// TIA Portal V17 export
// export: Created 2024-09-27T18:53:46.9042385Z, ExportSetting WithDefaults, DisplayName Totally Integrated Automation Portal, DisplayVersion V17, DisplayName TIA Portal Openness, DisplayVersion V17, DisplayName TIA Portal Version Control Interface, DisplayVersion V17, DisplayName STEP 7 Professional, DisplayVersion V17, DisplayName STEP 7 Safety, DisplayVersion V17, DisplayName WinCC Professional, DisplayVersion V17
FUNCTION "AUTOMAT" : Void   // FC6, LAD
{ S7_Optimized_Access := 'TRUE' }
VERSION : 0.1
// stored: AutoNumber true, IsIECCheckEnabled false, SetENOAutomatically false, UDAEnableTagReadback false
   VAR_TEMP
      m_zbocze_czujnik_poz_odb_stoł : Bool;
      m_zbocze_czujnik_stołP : Bool;
      m_zboczeN_czuj_plyt_przód : Bool;
      m_memo_stol_poz : Bool;
   END_VAR
   VAR_TEMP   // added for the SCL form of the ladder/FBD networks
      _w1 : Bool;
      _w2 : Bool;
   END_VAR
BEGIN

REGION Network 1: CHECK SERVO CONDITIONS
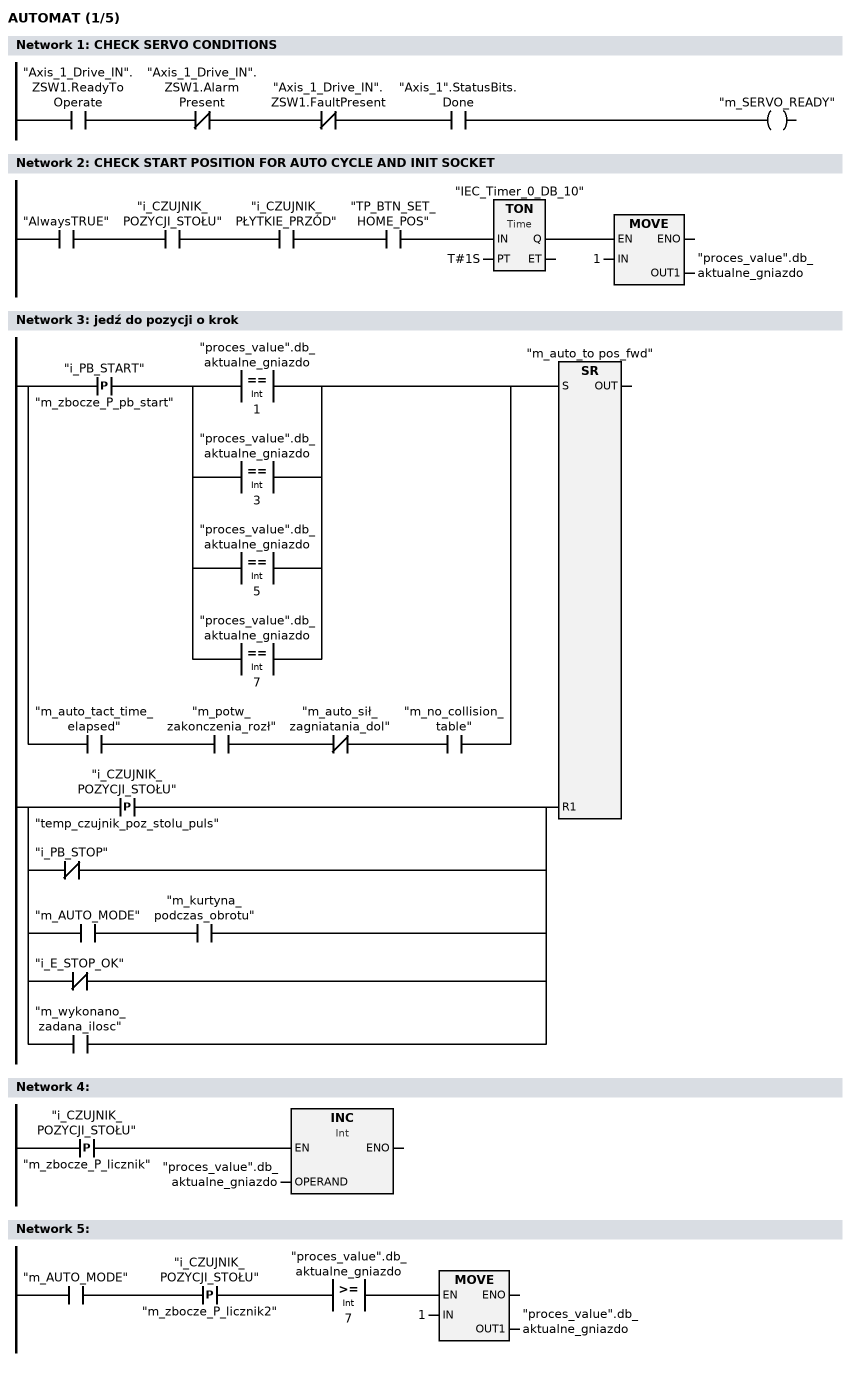
   RUNG wire#powerrail
      Contact( "Axis_1_Drive_IN".ZSW1.ReadyToOperate )
      I_Contact( "Axis_1_Drive_IN".ZSW1.AlarmPresent )
      I_Contact( "Axis_1_Drive_IN".ZSW1.FaultPresent )
      Contact( "Axis_1".StatusBits.Done )
      Coil( "m_SERVO_READY" )
   END_RUNG
   // the same network as SCL:
   "m_SERVO_READY" := "Axis_1_Drive_IN".ZSW1.ReadyToOperate AND NOT "Axis_1_Drive_IN".ZSW1.AlarmPresent AND NOT "Axis_1_Drive_IN".ZSW1.FaultPresent AND "Axis_1".StatusBits.Done;
END_REGION

REGION Network 2: CHECK START POSITION FOR AUTO CYCLE AND INIT SOCKET
   RUNG wire#powerrail
      Contact( "AlwaysTRUE" )
      Contact( "i_CZUJNIK_POZYCJI_STOŁU" )
      Contact( "i_CZUJNIK_PŁYTKIE_PRZÓD" )
      Contact( "TP_BTN_SET_HOME_POS" )
      { S7_Templates := "time_type := Time" } "IEC_Timer_0_DB_10".TON(pt := T#1S, et =>)
      Move(in := 1, out1 => "proces_value".db_aktualne_gniazdo)
   END_RUNG
   // the same network as SCL:
   "IEC_Timer_0_DB_10".TON(IN := "AlwaysTRUE" AND "i_CZUJNIK_POZYCJI_STOŁU" AND "i_CZUJNIK_PŁYTKIE_PRZÓD" AND "TP_BTN_SET_HOME_POS",
                           PT := T#1S);
   IF "IEC_Timer_0_DB_10".Q THEN "proces_value".db_aktualne_gniazdo := 1; END_IF;
END_REGION

REGION Network 3: jedź do pozycji o krok
   RUNG wire#powerrail
      P_Contact(operand := "i_PB_START", bit := "m_zbocze_P_pb_start")
      wire#w1
      { S7_Templates := "SrcType := Int" } EQ_Contact(in1 := "proces_value".db_aktualne_gniazdo, in2 := 1)
      wire#w2
      S_SR(operand := "m_auto_to pos_fwd", r1 := wire#w3)
   END_RUNG
   RUNG wire#w1
      { S7_Templates := "SrcType := Int" } EQ_Contact(in1 := "proces_value".db_aktualne_gniazdo, in2 := 3)
   END_RUNG wire#w2
   RUNG wire#w1
      { S7_Templates := "SrcType := Int" } EQ_Contact(in1 := "proces_value".db_aktualne_gniazdo, in2 := 5)
   END_RUNG wire#w2
   RUNG wire#w1
      { S7_Templates := "SrcType := Int" } EQ_Contact(in1 := "proces_value".db_aktualne_gniazdo, in2 := 7)
   END_RUNG wire#w2
   RUNG wire#powerrail
      Contact( "m_auto_tact_time_elapsed" )
      Contact( "m_potw_zakonczenia_rozł" )
      I_Contact( "m_auto_sił_zagniatania_dol" )
      Contact( "m_no_collision_table" )
   END_RUNG wire#w2
   RUNG wire#powerrail
      P_Contact(operand := "i_CZUJNIK_POZYCJI_STOŁU", bit := "temp_czujnik_poz_stolu_puls")
   END_RUNG wire#w3
   RUNG wire#powerrail
      I_Contact( "i_PB_STOP" )
   END_RUNG wire#w3
   RUNG wire#powerrail
      Contact( "m_AUTO_MODE" )
      Contact( "m_kurtyna_podczas_obrotu" )
   END_RUNG wire#w3
   RUNG wire#powerrail
      I_Contact( "i_E_STOP_OK" )
   END_RUNG wire#w3
   RUNG wire#powerrail
      Contact( "m_wykonano_zadana_ilosc" )
   END_RUNG wire#w3
   // the same network as SCL:
   #_w1 := "i_PB_START" AND NOT "m_zbocze_P_pb_start";   // rising edge of "i_PB_START"
   "m_zbocze_P_pb_start" := "i_PB_START";
   #_w2 := "i_CZUJNIK_POZYCJI_STOŁU" AND NOT "temp_czujnik_poz_stolu_puls";   // rising edge of "i_CZUJNIK_POZYCJI_STOŁU"
   "temp_czujnik_poz_stolu_puls" := "i_CZUJNIK_POZYCJI_STOŁU";
   IF (#_w1 AND (("proces_value".db_aktualne_gniazdo = 1) OR ("proces_value".db_aktualne_gniazdo = 3) OR ("proces_value".db_aktualne_gniazdo = 5) OR ("proces_value".db_aktualne_gniazdo = 7))) OR ("m_auto_tact_time_elapsed" AND "m_potw_zakonczenia_rozł" AND NOT "m_auto_sił_zagniatania_dol" AND "m_no_collision_table") THEN
       "m_auto_to pos_fwd" := TRUE;   // SR flip-flop
   END_IF;
   IF #_w2 OR NOT "i_PB_STOP" OR ("m_AUTO_MODE" AND "m_kurtyna_podczas_obrotu") OR NOT "i_E_STOP_OK" OR "m_wykonano_zadana_ilosc" THEN
       "m_auto_to pos_fwd" := FALSE;
   END_IF;
END_REGION

REGION Network 4
   RUNG wire#powerrail
      P_Contact(operand := "i_CZUJNIK_POZYCJI_STOŁU", bit := "m_zbocze_P_licznik")
      { S7_Templates := "DestType := Int" } Inc( "proces_value".db_aktualne_gniazdo )
   END_RUNG
   // the same network as SCL:
   #_w1 := "i_CZUJNIK_POZYCJI_STOŁU" AND NOT "m_zbocze_P_licznik";   // rising edge of "i_CZUJNIK_POZYCJI_STOŁU"
   "m_zbocze_P_licznik" := "i_CZUJNIK_POZYCJI_STOŁU";
   IF #_w1 THEN "proces_value".db_aktualne_gniazdo := "proces_value".db_aktualne_gniazdo + 1; END_IF;
END_REGION

REGION Network 5
   RUNG wire#powerrail
      Contact( "m_AUTO_MODE" )
      P_Contact(operand := "i_CZUJNIK_POZYCJI_STOŁU", bit := "m_zbocze_P_licznik2")
      { S7_Templates := "SrcType := Int" } GE_Contact(in1 := "proces_value".db_aktualne_gniazdo, in2 := 7)
      Move(in := 1, out1 => "proces_value".db_aktualne_gniazdo)
   END_RUNG
   // the same network as SCL:
   #_w1 := "m_AUTO_MODE" AND "i_CZUJNIK_POZYCJI_STOŁU" AND NOT "m_zbocze_P_licznik2";   // rising edge of "i_CZUJNIK_POZYCJI_STOŁU"
   "m_zbocze_P_licznik2" := "i_CZUJNIK_POZYCJI_STOŁU";
   IF #_w1 AND ("proces_value".db_aktualne_gniazdo >= 7) THEN
       "proces_value".db_aktualne_gniazdo := 1;
   END_IF;
END_REGION

REGION Network 6: zwłoka taktu
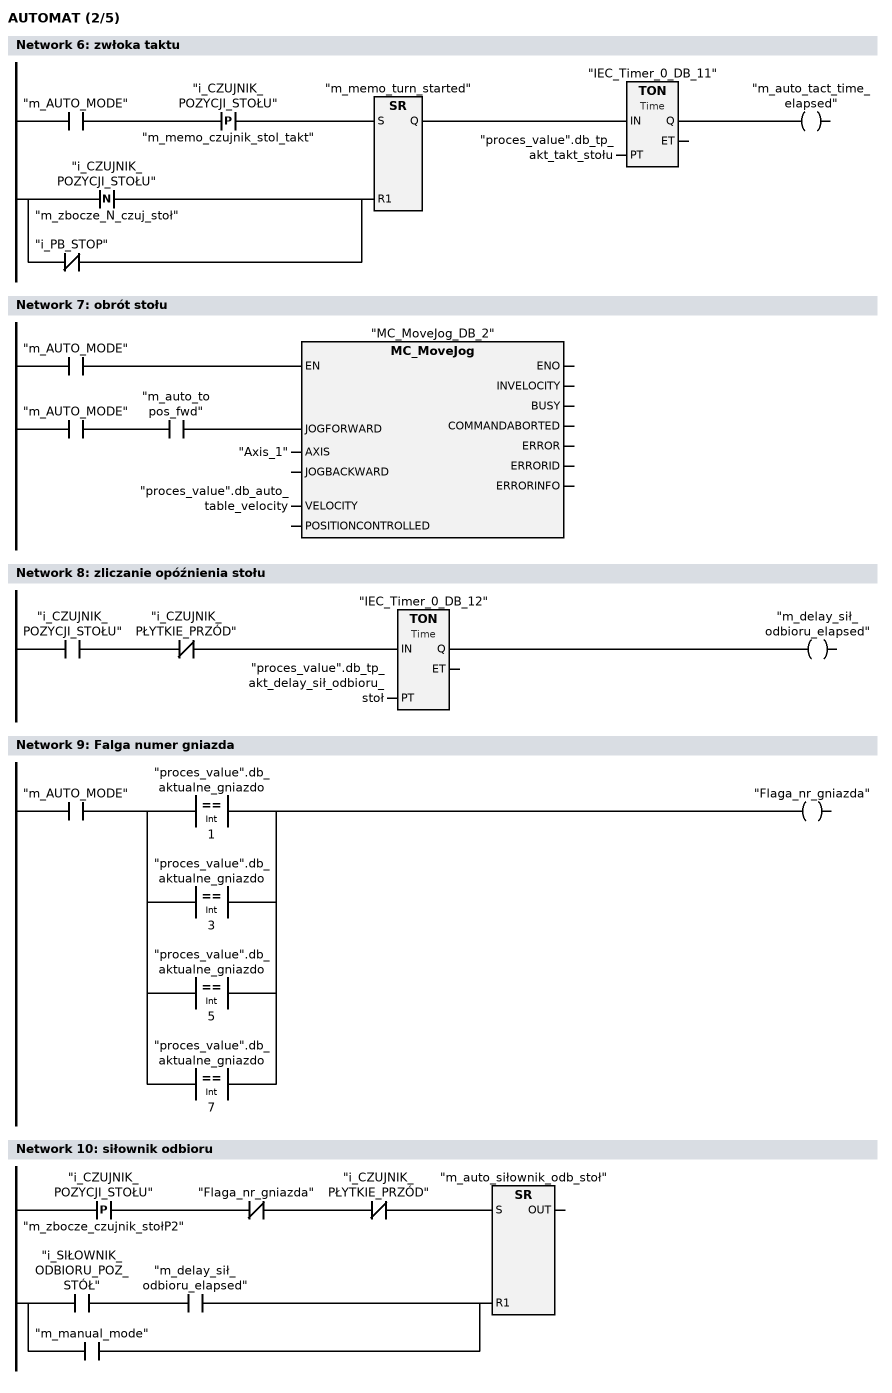
   RUNG wire#powerrail
      Contact( "m_AUTO_MODE" )
      P_Contact(operand := "i_CZUJNIK_POZYCJI_STOŁU", bit := "m_memo_czujnik_stol_takt")
      S_SR(operand := "m_memo_turn_started", r1 := wire#w1)
      { S7_Templates := "time_type := Time" } "IEC_Timer_0_DB_11".TON(pt := "proces_value".db_tp_akt_takt_stołu, et =>)
      Coil( "m_auto_tact_time_elapsed" )
   END_RUNG
   RUNG wire#powerrail
      N_Contact(operand := "i_CZUJNIK_POZYCJI_STOŁU", bit := "m_zbocze_N_czuj_stoł")
   END_RUNG wire#w1
   RUNG wire#powerrail
      I_Contact( "i_PB_STOP" )
   END_RUNG wire#w1
   // the same network as SCL:
   #_w1 := "m_AUTO_MODE" AND "i_CZUJNIK_POZYCJI_STOŁU" AND NOT "m_memo_czujnik_stol_takt";   // rising edge of "i_CZUJNIK_POZYCJI_STOŁU"
   "m_memo_czujnik_stol_takt" := "i_CZUJNIK_POZYCJI_STOŁU";
   #_w2 := NOT "i_CZUJNIK_POZYCJI_STOŁU" AND "m_zbocze_N_czuj_stoł";   // falling edge of "i_CZUJNIK_POZYCJI_STOŁU"
   "m_zbocze_N_czuj_stoł" := "i_CZUJNIK_POZYCJI_STOŁU";
   IF #_w1 THEN
       "m_memo_turn_started" := TRUE;   // SR flip-flop
   END_IF;
   IF #_w2 OR NOT "i_PB_STOP" THEN "m_memo_turn_started" := FALSE; END_IF;
   "IEC_Timer_0_DB_11".TON(IN := "m_memo_turn_started", PT := "proces_value".db_tp_akt_takt_stołu);
   "m_auto_tact_time_elapsed" := "IEC_Timer_0_DB_11".Q;
END_REGION

REGION Network 7: obrót stołu
   RUNG wire#powerrail
      Contact( "m_AUTO_MODE" )
      "MC_MoveJog_DB_2".MC_MoveJog(JogForward := wire#w1, Axis := "Axis_1", JogBackward :=, Velocity := "proces_value".db_auto_table_velocity, PositionControlled :=, InVelocity =>, Busy =>, CommandAborted =>, Error =>, ErrorID =>, ErrorInfo =>)
   END_RUNG
   RUNG wire#powerrail
      Contact( "m_AUTO_MODE" )
      Contact( "m_auto_to pos_fwd" )
   END_RUNG wire#w1
   // the same network as SCL:
   IF "m_AUTO_MODE" THEN
       "MC_MoveJog_DB_2"(JogForward := "m_AUTO_MODE" AND "m_auto_to pos_fwd",   // MC_MoveJog
                         Axis := "Axis_1",
                         Velocity := "proces_value".db_auto_table_velocity);
   END_IF;
END_REGION

REGION Network 8: zliczanie opóźnienia stołu
   RUNG wire#powerrail
      Contact( "i_CZUJNIK_POZYCJI_STOŁU" )
      I_Contact( "i_CZUJNIK_PŁYTKIE_PRZÓD" )
      { S7_Templates := "time_type := Time" } "IEC_Timer_0_DB_12".TON(pt := "proces_value".db_tp_akt_delay_sił_odbioru_stoł, et =>)
      Coil( "m_delay_sił_odbioru_elapsed" )
   END_RUNG
   // the same network as SCL:
   "IEC_Timer_0_DB_12".TON(IN := "i_CZUJNIK_POZYCJI_STOŁU" AND NOT "i_CZUJNIK_PŁYTKIE_PRZÓD",
                           PT := "proces_value".db_tp_akt_delay_sił_odbioru_stoł);
   "m_delay_sił_odbioru_elapsed" := "IEC_Timer_0_DB_12".Q;
END_REGION

REGION Network 9: Falga numer gniazda
   RUNG wire#powerrail
      Contact( "m_AUTO_MODE" )
      wire#w1
      { S7_Templates := "SrcType := Int" } EQ_Contact(in1 := "proces_value".db_aktualne_gniazdo, in2 := 1)
      wire#w2
      Coil( "Flaga_nr_gniazda" )
   END_RUNG
   RUNG wire#w1
      { S7_Templates := "SrcType := Int" } EQ_Contact(in1 := "proces_value".db_aktualne_gniazdo, in2 := 3)
   END_RUNG wire#w2
   RUNG wire#w1
      { S7_Templates := "SrcType := Int" } EQ_Contact(in1 := "proces_value".db_aktualne_gniazdo, in2 := 5)
   END_RUNG wire#w2
   RUNG wire#w1
      { S7_Templates := "SrcType := Int" } EQ_Contact(in1 := "proces_value".db_aktualne_gniazdo, in2 := 7)
   END_RUNG wire#w2
   // the same network as SCL:
   "Flaga_nr_gniazda" := "m_AUTO_MODE" AND (("proces_value".db_aktualne_gniazdo = 1) OR ("proces_value".db_aktualne_gniazdo = 3) OR ("proces_value".db_aktualne_gniazdo = 5) OR ("proces_value".db_aktualne_gniazdo = 7));
END_REGION

REGION Network 10: siłownik odbioru
   RUNG wire#powerrail
      P_Contact(operand := "i_CZUJNIK_POZYCJI_STOŁU", bit := "m_zbocze_czujnik_stołP2")
      I_Contact( "Flaga_nr_gniazda" )
      I_Contact( "i_CZUJNIK_PŁYTKIE_PRZÓD" )
      S_SR(operand := "m_auto_siłownik_odb_stoł", r1 := wire#w1)
   END_RUNG
   RUNG wire#powerrail
      Contact( "i_SIŁOWNIK_ODBIORU_POZ_STÓŁ" )
      Contact( "m_delay_sił_odbioru_elapsed" )
   END_RUNG wire#w1
   RUNG wire#powerrail
      Contact( "m_manual_mode" )
   END_RUNG wire#w1
   // the same network as SCL:
   #_w1 := "i_CZUJNIK_POZYCJI_STOŁU" AND NOT "m_zbocze_czujnik_stołP2";   // rising edge of "i_CZUJNIK_POZYCJI_STOŁU"
   "m_zbocze_czujnik_stołP2" := "i_CZUJNIK_POZYCJI_STOŁU";
   IF #_w1 AND NOT "Flaga_nr_gniazda" AND NOT "i_CZUJNIK_PŁYTKIE_PRZÓD" THEN
       "m_auto_siłownik_odb_stoł" := TRUE;   // SR flip-flop
   END_IF;
   IF ("i_SIŁOWNIK_ODBIORU_POZ_STÓŁ" AND "m_delay_sił_odbioru_elapsed") OR "m_manual_mode" THEN
       "m_auto_siłownik_odb_stoł" := FALSE;
   END_IF;
END_REGION

REGION Network 11
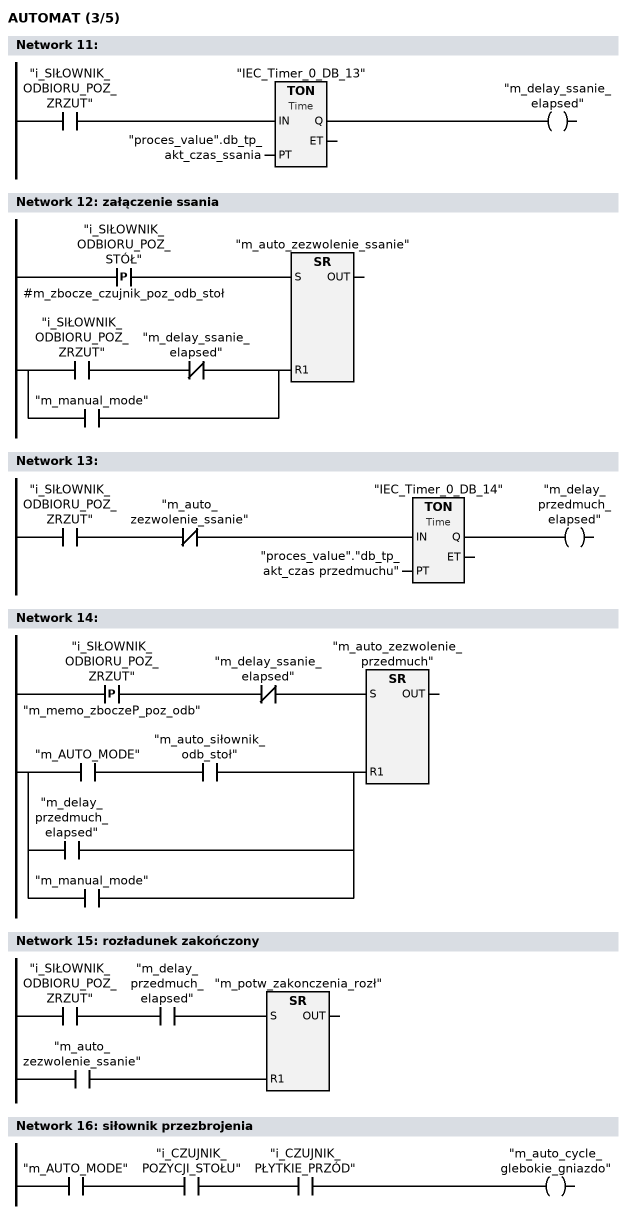
   RUNG wire#powerrail
      Contact( "i_SIŁOWNIK_ODBIORU_POZ_ZRZUT" )
      { S7_Templates := "time_type := Time" } "IEC_Timer_0_DB_13".TON(pt := "proces_value".db_tp_akt_czas_ssania, et =>)
      Coil( "m_delay_ssanie_elapsed" )
   END_RUNG
   // the same network as SCL:
   "IEC_Timer_0_DB_13".TON(IN := "i_SIŁOWNIK_ODBIORU_POZ_ZRZUT", PT := "proces_value".db_tp_akt_czas_ssania);
   "m_delay_ssanie_elapsed" := "IEC_Timer_0_DB_13".Q;
END_REGION

REGION Network 12: załączenie ssania
   RUNG wire#powerrail
      P_Contact(operand := "i_SIŁOWNIK_ODBIORU_POZ_STÓŁ", bit := #m_zbocze_czujnik_poz_odb_stoł)
      S_SR(operand := "m_auto_zezwolenie_ssanie", r1 := wire#w1)
   END_RUNG
   RUNG wire#powerrail
      Contact( "i_SIŁOWNIK_ODBIORU_POZ_ZRZUT" )
      I_Contact( "m_delay_ssanie_elapsed" )
   END_RUNG wire#w1
   RUNG wire#powerrail
      Contact( "m_manual_mode" )
   END_RUNG wire#w1
   // the same network as SCL:
   #_w1 := "i_SIŁOWNIK_ODBIORU_POZ_STÓŁ" AND NOT #m_zbocze_czujnik_poz_odb_stoł;   // rising edge of "i_SIŁOWNIK_ODBIORU_POZ_STÓŁ"
   #m_zbocze_czujnik_poz_odb_stoł := "i_SIŁOWNIK_ODBIORU_POZ_STÓŁ";
   IF #_w1 THEN
       "m_auto_zezwolenie_ssanie" := TRUE;   // SR flip-flop
   END_IF;
   IF ("i_SIŁOWNIK_ODBIORU_POZ_ZRZUT" AND NOT "m_delay_ssanie_elapsed") OR "m_manual_mode" THEN
       "m_auto_zezwolenie_ssanie" := FALSE;
   END_IF;
END_REGION

REGION Network 13
   RUNG wire#powerrail
      Contact( "i_SIŁOWNIK_ODBIORU_POZ_ZRZUT" )
      I_Contact( "m_auto_zezwolenie_ssanie" )
      { S7_Templates := "time_type := Time" } "IEC_Timer_0_DB_14".TON(pt := "proces_value"."db_tp_akt_czas przedmuchu", et =>)
      Coil( "m_delay_przedmuch_elapsed" )
   END_RUNG
   // the same network as SCL:
   "IEC_Timer_0_DB_14".TON(IN := "i_SIŁOWNIK_ODBIORU_POZ_ZRZUT" AND NOT "m_auto_zezwolenie_ssanie",
                           PT := "proces_value"."db_tp_akt_czas przedmuchu");
   "m_delay_przedmuch_elapsed" := "IEC_Timer_0_DB_14".Q;
END_REGION

REGION Network 14
   RUNG wire#powerrail
      P_Contact(operand := "i_SIŁOWNIK_ODBIORU_POZ_ZRZUT", bit := "m_memo_zboczeP_poz_odb")
      I_Contact( "m_delay_ssanie_elapsed" )
      S_SR(operand := "m_auto_zezwolenie_przedmuch", r1 := wire#w1)
   END_RUNG
   RUNG wire#powerrail
      Contact( "m_AUTO_MODE" )
      Contact( "m_auto_siłownik_odb_stoł" )
   END_RUNG wire#w1
   RUNG wire#powerrail
      Contact( "m_delay_przedmuch_elapsed" )
   END_RUNG wire#w1
   RUNG wire#powerrail
      Contact( "m_manual_mode" )
   END_RUNG wire#w1
   // the same network as SCL:
   #_w1 := "i_SIŁOWNIK_ODBIORU_POZ_ZRZUT" AND NOT "m_memo_zboczeP_poz_odb";   // rising edge of "i_SIŁOWNIK_ODBIORU_POZ_ZRZUT"
   "m_memo_zboczeP_poz_odb" := "i_SIŁOWNIK_ODBIORU_POZ_ZRZUT";
   IF #_w1 AND NOT "m_delay_ssanie_elapsed" THEN
       "m_auto_zezwolenie_przedmuch" := TRUE;   // SR flip-flop
   END_IF;
   IF ("m_AUTO_MODE" AND "m_auto_siłownik_odb_stoł") OR "m_delay_przedmuch_elapsed" OR "m_manual_mode" THEN
       "m_auto_zezwolenie_przedmuch" := FALSE;
   END_IF;
END_REGION

REGION Network 15: rozładunek zakończony
   RUNG wire#powerrail
      Contact( "i_SIŁOWNIK_ODBIORU_POZ_ZRZUT" )
      Contact( "m_delay_przedmuch_elapsed" )
      S_SR(operand := "m_potw_zakonczenia_rozł", r1 := wire#w1)
   END_RUNG
   RUNG wire#powerrail
      Contact( "m_auto_zezwolenie_ssanie" )
   END_RUNG wire#w1
   // the same network as SCL:
   IF "i_SIŁOWNIK_ODBIORU_POZ_ZRZUT" AND "m_delay_przedmuch_elapsed" THEN
       "m_potw_zakonczenia_rozł" := TRUE;   // SR flip-flop
   END_IF;
   IF "m_auto_zezwolenie_ssanie" THEN "m_potw_zakonczenia_rozł" := FALSE; END_IF;
END_REGION

REGION Network 16: siłownik przezbrojenia
   RUNG wire#powerrail
      Contact( "m_AUTO_MODE" )
      Contact( "i_CZUJNIK_POZYCJI_STOŁU" )
      Contact( "i_CZUJNIK_PŁYTKIE_PRZÓD" )
      Coil( "m_auto_cycle_glebokie_gniazdo" )
   END_RUNG
   // the same network as SCL:
   "m_auto_cycle_glebokie_gniazdo" := "m_AUTO_MODE" AND "i_CZUJNIK_POZYCJI_STOŁU" AND "i_CZUJNIK_PŁYTKIE_PRZÓD";
END_REGION

REGION Network 17: Interlock na zmiane podczas ruchu siłownika góra dół
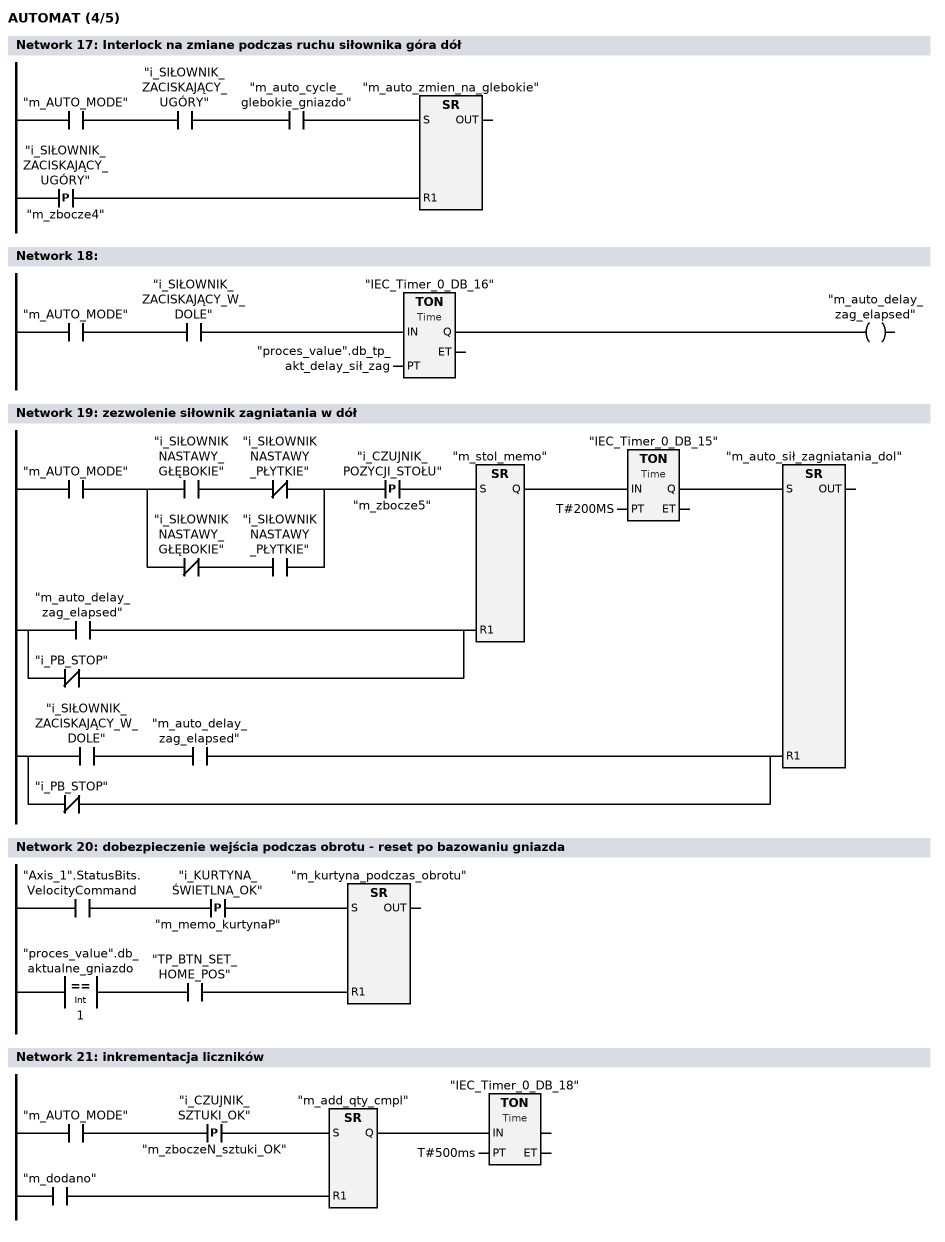
   RUNG wire#powerrail
      Contact( "m_AUTO_MODE" )
      Contact( "i_SIŁOWNIK_ZACISKAJĄCY_UGÓRY" )
      Contact( "m_auto_cycle_glebokie_gniazdo" )
      S_SR(operand := "m_auto_zmien_na_glebokie", r1 := wire#w1)
   END_RUNG
   RUNG wire#powerrail
      P_Contact(operand := "i_SIŁOWNIK_ZACISKAJĄCY_UGÓRY", bit := "m_zbocze4")
   END_RUNG wire#w1
   // the same network as SCL:
   #_w1 := "i_SIŁOWNIK_ZACISKAJĄCY_UGÓRY" AND NOT "m_zbocze4";   // rising edge of "i_SIŁOWNIK_ZACISKAJĄCY_UGÓRY"
   "m_zbocze4" := "i_SIŁOWNIK_ZACISKAJĄCY_UGÓRY";
   IF "m_AUTO_MODE" AND "i_SIŁOWNIK_ZACISKAJĄCY_UGÓRY" AND "m_auto_cycle_glebokie_gniazdo" THEN
       "m_auto_zmien_na_glebokie" := TRUE;   // SR flip-flop
   END_IF;
   IF #_w1 THEN "m_auto_zmien_na_glebokie" := FALSE; END_IF;
END_REGION

REGION Network 18
   RUNG wire#powerrail
      Contact( "m_AUTO_MODE" )
      Contact( "i_SIŁOWNIK_ZACISKAJĄCY_W_DOLE" )
      { S7_Templates := "time_type := Time" } "IEC_Timer_0_DB_16".TON(pt := "proces_value".db_tp_akt_delay_sił_zag, et =>)
      Coil( "m_auto_delay_zag_elapsed" )
   END_RUNG
   // the same network as SCL:
   "IEC_Timer_0_DB_16".TON(IN := "m_AUTO_MODE" AND "i_SIŁOWNIK_ZACISKAJĄCY_W_DOLE",
                           PT := "proces_value".db_tp_akt_delay_sił_zag);
   "m_auto_delay_zag_elapsed" := "IEC_Timer_0_DB_16".Q;
END_REGION

REGION Network 19: zezwolenie siłownik zagniatania w dół
   RUNG wire#powerrail
      Contact( "m_AUTO_MODE" )
      wire#w1
      Contact( "i_SIŁOWNIK NASTAWY_GŁĘBOKIE" )
      I_Contact( "i_SIŁOWNIK NASTAWY _PŁYTKIE" )
      wire#w2
      P_Contact(operand := "i_CZUJNIK_POZYCJI_STOŁU", bit := "m_zbocze5")
      S_SR(operand := "m_stol_memo", r1 := wire#w3)
      { S7_Templates := "time_type := Time" } "IEC_Timer_0_DB_15".TON(pt := T#200MS, et =>)
      S_SR(operand := "m_auto_sił_zagniatania_dol", r1 := wire#w4)
   END_RUNG
   RUNG wire#w1
      I_Contact( "i_SIŁOWNIK NASTAWY_GŁĘBOKIE" )
      Contact( "i_SIŁOWNIK NASTAWY _PŁYTKIE" )
   END_RUNG wire#w2
   RUNG wire#powerrail
      Contact( "m_auto_delay_zag_elapsed" )
   END_RUNG wire#w3
   RUNG wire#powerrail
      I_Contact( "i_PB_STOP" )
   END_RUNG wire#w3
   RUNG wire#powerrail
      Contact( "i_SIŁOWNIK_ZACISKAJĄCY_W_DOLE" )
      Contact( "m_auto_delay_zag_elapsed" )
   END_RUNG wire#w4
   RUNG wire#powerrail
      I_Contact( "i_PB_STOP" )
   END_RUNG wire#w4
   // the same network as SCL:
   #_w1 := "m_AUTO_MODE" AND (("i_SIŁOWNIK NASTAWY_GŁĘBOKIE" AND NOT "i_SIŁOWNIK NASTAWY _PŁYTKIE") OR (NOT "i_SIŁOWNIK NASTAWY_GŁĘBOKIE" AND "i_SIŁOWNIK NASTAWY _PŁYTKIE")) AND "i_CZUJNIK_POZYCJI_STOŁU" AND NOT "m_zbocze5";   // rising edge of "i_CZUJNIK_POZYCJI_STOŁU"
   "m_zbocze5" := "i_CZUJNIK_POZYCJI_STOŁU";
   IF #_w1 THEN
       "m_stol_memo" := TRUE;   // SR flip-flop
   END_IF;
   IF "m_auto_delay_zag_elapsed" OR NOT "i_PB_STOP" THEN "m_stol_memo" := FALSE; END_IF;
   "IEC_Timer_0_DB_15".TON(IN := "m_stol_memo", PT := T#200MS);
   IF "IEC_Timer_0_DB_15".Q THEN
       "m_auto_sił_zagniatania_dol" := TRUE;   // SR flip-flop
   END_IF;
   IF ("i_SIŁOWNIK_ZACISKAJĄCY_W_DOLE" AND "m_auto_delay_zag_elapsed") OR NOT "i_PB_STOP" THEN
       "m_auto_sił_zagniatania_dol" := FALSE;
   END_IF;
END_REGION

REGION Network 20: dobezpieczenie wejścia podczas obrotu - reset po bazowaniu gniazda
   RUNG wire#powerrail
      Contact( "Axis_1".StatusBits.VelocityCommand )
      P_Contact(operand := "i_KURTYNA_ŚWIETLNA_OK", bit := "m_memo_kurtynaP")
      S_SR(operand := "m_kurtyna_podczas_obrotu", r1 := wire#w1)
   END_RUNG
   RUNG wire#powerrail
      { S7_Templates := "SrcType := Int" } EQ_Contact(in1 := "proces_value".db_aktualne_gniazdo, in2 := 1)
      Contact( "TP_BTN_SET_HOME_POS" )
   END_RUNG wire#w1
   // the same network as SCL:
   #_w1 := "Axis_1".StatusBits.VelocityCommand AND "i_KURTYNA_ŚWIETLNA_OK" AND NOT "m_memo_kurtynaP";   // rising edge of "i_KURTYNA_ŚWIETLNA_OK"
   "m_memo_kurtynaP" := "i_KURTYNA_ŚWIETLNA_OK";
   IF #_w1 THEN
       "m_kurtyna_podczas_obrotu" := TRUE;   // SR flip-flop
   END_IF;
   IF ("proces_value".db_aktualne_gniazdo = 1) AND "TP_BTN_SET_HOME_POS" THEN
       "m_kurtyna_podczas_obrotu" := FALSE;
   END_IF;
END_REGION

REGION Network 21: inkrementacja liczników
   RUNG wire#powerrail
      Contact( "m_AUTO_MODE" )
      P_Contact(operand := "i_CZUJNIK_SZTUKI_OK", bit := "m_zboczeN_sztuki_OK")
      S_SR(operand := "m_add_qty_cmpl", r1 := wire#w1)
      { S7_Templates := "time_type := Time" } "IEC_Timer_0_DB_18".TON(pt := T#500ms, et =>)
   END_RUNG
   RUNG wire#powerrail
      Contact( "m_dodano" )
   END_RUNG wire#w1
   // the same network as SCL:
   #_w1 := "m_AUTO_MODE" AND "i_CZUJNIK_SZTUKI_OK" AND NOT "m_zboczeN_sztuki_OK";   // rising edge of "i_CZUJNIK_SZTUKI_OK"
   "m_zboczeN_sztuki_OK" := "i_CZUJNIK_SZTUKI_OK";
   IF #_w1 THEN
       "m_add_qty_cmpl" := TRUE;   // SR flip-flop
   END_IF;
   IF "m_dodano" THEN "m_add_qty_cmpl" := FALSE; END_IF;
   "IEC_Timer_0_DB_18".TON(IN := "m_add_qty_cmpl", PT := T#500ms);
END_REGION

REGION Network 22
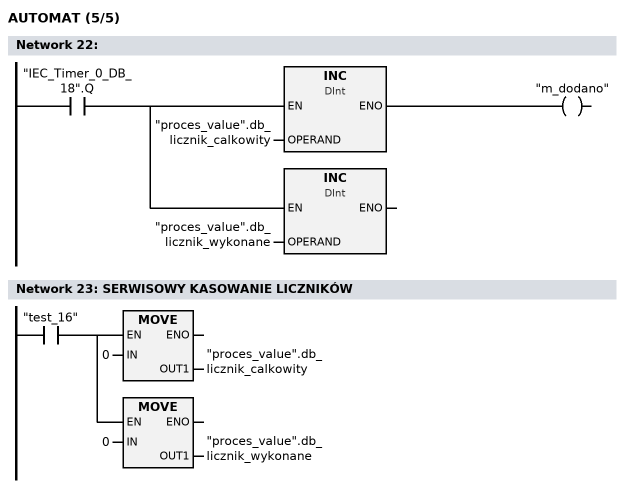
   RUNG wire#powerrail
      Contact( "IEC_Timer_0_DB_18".Q )
      wire#w1
      { S7_Templates := "DestType := DInt" } Inc( "proces_value".db_licznik_calkowity )
      Coil( "m_dodano" )
   END_RUNG
   RUNG wire#w1
      { S7_Templates := "DestType := DInt" } Inc( "proces_value".db_licznik_wykonane )
   END_RUNG
   // the same network as SCL:
   IF "IEC_Timer_0_DB_18".Q THEN
       "proces_value".db_licznik_calkowity := "proces_value".db_licznik_calkowity + 1;
   END_IF;
   "m_dodano" := "IEC_Timer_0_DB_18".Q;
   IF "IEC_Timer_0_DB_18".Q THEN
       "proces_value".db_licznik_wykonane := "proces_value".db_licznik_wykonane + 1;
   END_IF;
END_REGION

REGION Network 23: SERWISOWY KASOWANIE LICZNIKÓW
   RUNG wire#powerrail
      Contact( "test_16" )
      wire#w1
      Move(in := 0, out1 => "proces_value".db_licznik_calkowity)
   END_RUNG
   RUNG wire#w1
      Move(in := 0, out1 => "proces_value".db_licznik_wykonane)
   END_RUNG
   // the same network as SCL:
   IF "test_16" THEN
       "proces_value".db_licznik_calkowity := 0;
       "proces_value".db_licznik_wykonane := 0;
   END_IF;
END_REGION
END_FUNCTION
